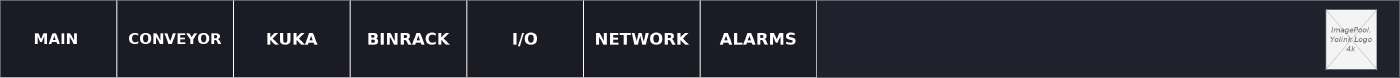
VISUALIZATION HEADER  // 1920x108
    Rectangle (0,0 1920x108)
    RoundedRectangle (0,0 160x108), "MAIN"
        OnMouseClick: change screen: MAIN_PAGE
    RoundedRectangle (160,0 160x108), "CONVEYOR"
        OnMouseClick: change screen: CONVEYOR_PAGE
    RoundedRectangle (320,0 160x108), "KUKA"
        OnMouseClick: change screen: KUKA_PAGE
    RoundedRectangle (480,0 160x108), "BINRACK"
        OnMouseClick: change screen: BINRACK_PAGE
    RoundedRectangle (640,0 160x108), "I/O"
        OnMouseClick: change screen: PLC_IO_PAGE
    RoundedRectangle (960,0 160x108), "ALARMS"
    RoundedRectangle (800,0 160x108), "NETWORK"
        OnMouseClick: change screen: NETWORK_PAGE
    Rectangle (1760,0 160x108), text variable: MAIN.fb_TimeStamp.SystemTime
    Textfield (1760,20 160x30), "%s", text variable: MAIN.fb_TimeStamp.SystemTime
    Textfield (1760,59 160x30), "%s", text variable: MAIN.fb_TimeStamp.SystemDate
    Image (1818,13 70x83), image: ImagePool.Yolink Logo 4k
END_VISUALIZATION

(* stored: Version 1.1.0.1, ProductVersion 3.1.4024.12
   Visu HEADER: Id {9b99c136-28e5-42bf-9f40-a007d747a887} *)
